PROGRAM MAIN
VAR
	
	status0:BOOL;
	
END_VAR

Alias();
CAN_comm();
Tx_MasterPLC();
//CanInterface();
AnalogConversion();
Permissives();
Trips();
MODE_SELECTION_1();
//Trips_LAD();
Alarms();
//Graphs();
Heartbeat();
VoltageOutputCal();
Cal_ChargeTime();


//test
//IF MCP_IO.AutoModeSelected THEN
//	Output.R2_05_07 := heartbeat.pulse_1Hz;
//END_IF

	
//sample test
IF gvl.test = TRUE THEN
	Output.R2_05_00 := TRUE;
	ELSE 
		Output.R2_05_00 := FALSE; 	
END_IF;

END_PROGRAM

(* stored: Version 1.1.0.1, ProductVersion 3.1.4024.11
   POU MAIN: Id {f38eb3b9-bd5e-4d40-a781-f42b0e7eec9a}, SpecialFunc None *)
